DATA_BLOCK "SelvMaGeneral_HMI"
{ S7_Optimized_Access := 'FALSE' }
VERSION : 0.1
   STRUCT
      tHMR : Struct   // {[Unit]|[Scada Unit]|[LowLimit]|[HigLimit]|[Acces]}
         xAutoDriftControlEnabled : Array["STARTARRAY".."DNUMSECTION"] of Bool;   // Auto Drift Control Enabled  {x|x|x|x|O}
         xAutoCapControlEnabled : Array["STARTARRAY".."DNUMSECTION"] of Bool;   // Auto Cap Widht Control Enabled  {x|x|x|x|O}
         xCulletEdgeEnabled : Bool;   // Cullet edge Enabled{x|x|x|x|O}
      END_STRUCT;
      tHMW : Struct   // {[Unit]|[Scada Unit]|[LowLimit]|[HigLimit]|[Acces]}
         xEnableDisableAutoDriftControl : Array["STARTARRAY".."DNUMSECTION"] of Bool;   // Enable Disable Auto Drift Control {x|x|x|x|O}
         xEnableDisableAutoCapControl : Array["STARTARRAY".."DNUMSECTION"] of Bool;   // Enable Disable Auto Cap Widht Control  {x|x|x|x|O}
         xEnableDisableCulletEdge : Bool;   // Enable Disable Cullet edge {x|x|x|x|O}
         xConfirmResetOffset : Bool;   // Confirm Reset offset {x|x|x|x|O}
         dWidhtCapForAutoContrloCapDisable_cmm : DInt;   // Widht For Auto Control Disable (work if you Auto Cap Control is disabled){cmm|cmm|x|x|O}
         dStepPushButtons_cmm : DInt;   // Step in cmm when press pushbuttons Offset
         rWidhtCapForAutoContrloCapDisable_mm : Real;   // Widht For Auto Control Disable (work if you Auto Cap Control is disabled){mm|mm|x|x|O}
         rStepPushButtons_mm : Real;   // Step in mm when press pushbuttons Offset
         tResetOffsetFr : Array["STARTARRAY".."DNUMFRAME"] of Bool;   // Reset offset Frame {x|x|x|x|O}
         tResetOffsetWhBrk : Array["STARTARRAY".."DNUMWHEEL"] of Bool;   // Reset offset Whell Brk {x|x|x|x|O}
      END_STRUCT;
   END_STRUCT;


BEGIN

END_DATA_BLOCK

